PROGRAM PRG_FB_BowlFeeder
VAR
	bFirstCycle 			: BOOL := TRUE;
	fbBowlFeeder 			: FB_BowlFeeder;
	
	rSetSp	: REAL := 50;

	bInit 					: BOOL;
	bAbort 					: BOOL;
	bReset					: BOOL;
	bStart					: BOOL;
	bStop					: BOOL;

	bActive					: BOOL;
	bRunning				: BOOL;
	bError					: BOOL;
	iErrorID				: UDINT;
	

	rSetpoint: REAL;
END_VAR

(* Setting initial parameters *)
IF bFirstCycle THEN
	bFirstCycle := FALSE;
	
	fbBowlFeeder.MR_FirstCycle(sName := 'Bowl Feeder');
	fbBowlFeeder.Setpoint := rSetSp;
END_IF

bActive := fbBowlFeeder.Active;
bRunning := fbBowlFeeder.Running;
bError := fbBowlFeeder.Error;
rSetpoint := fbBowlFeeder.Setpoint;

(* Simple controler *)
IF bInit THEN
	fbBowlFeeder.MR_Init();
	IF fbBowlFeeder.Active THEN
		bInit := FALSE;
	END_IF
END_IF

IF bStart THEN
	fbBowlFeeder.MR_Start();
	IF fbBowlFeeder.Running THEN
 		bStart := FALSE;
	END_IF
END_IF

IF bStop THEN
	fbBowlFeeder.MR_Stop();
	IF NOT fbBowlFeeder.Running THEN
 		bStop := FALSE;
	END_IF
END_IF

fbBowlFeeder();

END_PROGRAM

(* stored: Version 1.1.0.1, ProductVersion 3.1.4024.9
   POU PRG_FB_BowlFeeder: Id {8c8ea1ee-d264-4438-888b-083a28ed0fdc}, SpecialFunc None *)
